// TwinCAT 3 PLC project TwinCAT_OpenFramework_Loggers
// Title: TwinCAT Open Framework Loggers
// Company: Oleksandr Tiutyk FOP
// Author: Oleksandr Tiutyk
// ProjectVersion: 1.0.13.0
// Description: Various loggers implementation for TwinCAT.OpenFramework
// ProgramVersion: 3.1.4026.28
// libraries:
//   Tc2_Standard, * (Beckhoff Automation GmbH)
//   Tc2_System, * (Beckhoff Automation GmbH)
//   Tc2_Utilities, * (Beckhoff Automation GmbH)
//   Tc3_EventLogger, * (Beckhoff Automation GmbH)
//   Tc3_Module, * (Beckhoff Automation GmbH)
//   [TwinCAT Open Framework Collections], * (Oleksandr Tiutyk FOP)
//   [TwinCAT Open Framework Core], * (Oleksandr Tiutyk FOP)
//   [TwinCAT Open Framework File System], * (Oleksandr Tiutyk FOP)
// project tree:
//   QueuedLogger/ QueuedLogger.TcPOU, QUEUED_LOG_MESSAGE.TcDUT
//   / Parameters.TcGVL
//   EventLogger/ EventLogger.TcPOU
//   FileLogger/ SimpleTextFileLogger.TcPOU, SIMPLE_TEXT_FILE_LOGGER_STATE.TcDUT
//   Internal/ CurrentNamespace.TcPOU, NamespaceExtractor.TcPOU
//   Version/ Global_Version.TcGVL
// (motion and I/O tree: see PLC project twincat_openframework_core)
// real-time tasks:
//   TASK PlcTask: cycle T#10ms, priority 20, ADS port 350
//   TASK TestTask: cycle T#10ms, priority 1, ADS port 351
//   TASK RunnerTestTask: cycle T#10ms, priority 2, ADS port 354
//   TASK HowToTask: cycle T#10ms, priority 22, ADS port 353
// variable links:

// ---- QueuedLogger/QUEUED_LOG_MESSAGE.TcDUT
(*
SPDX-FileCopyrightText: © 2026 Oleksandr Tiutyk <trofimich@gmail.com>
SPDX-License-Identifier: MIT
License: https://opensource.org/license/mit
*)

(*!
<summary>Stores an owned text snapshot waiting for a logging backend.</summary>
<description>
Internal QueuedLogger storage. Text, category and optional number are copied by value. Contains no borrowed
references to caller data or exceptions.
</description>
*)
TYPE QUEUED_LOG_MESSAGE :
STRUCT
	Message : TOF_Core.ERROR_MESSAGE;
	Category : TOF_Core.LOG_CATEGORY;
	HasMessageNumber : BOOL;
	MessageNumber : ULINT;
END_STRUCT
END_TYPE

// ---- FileLogger/SIMPLE_TEXT_FILE_LOGGER_STATE.TcDUT
(*!
<summary>Identifies the current phase of a text-file logger.</summary>
<description>
Stop first drains accepted messages in the current initialization/logging phase. STOPPING then advances final
file release; STOPPED permits explicit Start. FAILED remains terminal and may still require cyclic cleanup.
New states follow FAILED so the existing state ordinals remain unchanged.
</description>
*)
{attribute 'qualified_only'}
{attribute 'strict'}
{attribute 'to_string'}
TYPE SIMPLE_TEXT_FILE_LOGGER_STATE :
(
	INITIAL,
	CREATING_DIRECTORY, 
	LOGGING, 
	FAILED,
	STOPPING,
	STOPPED
);
END_TYPE

// ---- Parameters.TcGVL
(*
SPDX-FileCopyrightText: © 2026 Oleksandr Tiutyk <trofimich@gmail.com>
SPDX-License-Identifier: MIT
License: https://opensource.org/license/mit
*)

(*!
<summary>Provides configurable library limits for logging.</summary>
<description>Limits apply independently to each logger instance, not to a shared memory budget.</description>
*)
{attribute 'qualified_only'}
VAR_GLOBAL CONSTANT
	(*!
	<summary>Maximum number of messages waiting in each SimpleTextFileLogger message queue.</summary>
	<description>
	When the queue reaches this limit, TryLog methods return FALSE before formatting or allocating queued text.
	Already accepted messages are retained. The current send batch is excluded and is limited separately by
	maxRecordsPerFile. Zero prevents acceptance of new messages.
	</description>
	*)
	MAX_PENDING_LOG_MESSAGES : UINT := 50;

	(*!
	<summary>Maximum number of text records waiting in each QueuedLogger.</summary>
	<description>
	Fixed per-instance storage; each record includes an ERROR_MESSAGE and number metadata. The array reserves one
	extra slot so zero capacity is representable; zero rejects all records. One additional record is reserved for
	the active backend call. Capacity also bounds records forwarded by one Execute. Full queues reject new
	records without waiting for free space; acquiring the queue lock may still block.
	</description>
	*)
	QUEUED_LOGGER_CAPACITY : UINT := 100;
END_VAR

// ---- Version/Global_Version.TcGVL
{attribute 'TcGenerated'}
{attribute 'no-analysis'}
{attribute 'linkalways'}
// This function has been automatically generated from the project information.
VAR_GLOBAL CONSTANT
	{attribute 'const_non_replaced'}
	stLibVersion_TwinCAT_Open_Framework_Loggers : ST_LibVersion := (iMajor := 1, iMinor := 0, iBuild := 13, iRevision := 0, nFlags := 0, sVersion := '1.0.13.0');
END_VAR

// ---- FileLogger/SimpleTextFileLogger.TcPOU
(*
SPDX-FileCopyrightText: © 2026 Oleksandr Tiutyk <trofimich@gmail.com>
SPDX-License-Identifier: MIT
License: https://opensource.org/license/mit
*)

(*!
<summary>Formats diagnostics for text-file logging and advances file operations through cyclic execution.</summary>
<description>
Use this backend for buffered text-file output. Direct TryLog and Execute calls on one instance must belong to
one task: its message queue, buffers and file-operation state are not synchronized for concurrent access. For
callers in multiple tasks, use QueuedLogger and let its owner task service this backend; do not bypass the
wrapper with concurrent direct calls. Separate instances writing independently must use separate output files.
Cyclic Execute is required to advance writing and cleanup. Exception logging accepts IReadOnlyException and
reads borrowed diagnostics without transferring ownership. Implementations must not retain exception
references beyond their task cleanup. FAILED is terminal for this instance: no automatic retry or recovery is
provided. Continue calling Execute after failure to discard queued messages, cancel active tasks and release
the send buffer once file operations have finished. Pending messages are not retried. The instance must remain
alive during cleanup. Busy reports pending initialization, messages, file operations or failure cleanup; an
idle open file alone does not make it TRUE. Busy = FALSE does not mean the file handle is closed. After Stop
or in FAILED state, or when the per-instance message queue reaches Parameters.MAX_PENDING_LOG_MESSAGES, all
TryLog methods return FALSE before formatting or queuing new diagnostics. Full-queue rejection preserves
already accepted messages; the current send batch is separate from this limit. Buffered text preserves the
optional message number and category prefix; oversized text is truncated to ERROR_MESSAGE capacity with a
final ellipsis. TryLog methods and Execute do not propagate exceptions. Failed admission returns FALSE;
Execute failures enter FAILED and require further cleanup calls. The terminal allocation latch is preserved
for the task boundary. The initial instance starts automatically through Execute. Stop requests draining of
accepted messages and best-effort file release; continue Execute until STOPPED or until FAILED cleanup
finishes. Start resumes only STOPPED, retaining the file counter and opening the next generated file when a
message arrives. New messages are rejected from Stop until Start. Lifecycle calls belong to the same owner
task as Execute. STOPPED means the close attempt and buffer cleanup finished, not certified physical closure
after a native close error; the underlying resource manager retains its best-effort policy. Embedded task
and resource diagnostics use an owned AdsLogger directly, bypassing LogManager filters/counters and avoiding
feedback into this logger or its QueuedLogger wrapper. maxRecordsPerFile must be positive; zero rejects
admission and the first Execute enters FAILED before any filesystem operation. The configured timeout
applies to directory, open, write and close requests, not to the whole logger lifecycle.
</description>
*)

{attribute 'no_explicit_call' := 'do not call this function block directly'}
FUNCTION_BLOCK SimpleTextFileLogger EXTENDS TOF_Core.Object IMPLEMENTS TOF_Core.ILogger
VAR_STAT
	//! <summary>Static type metadata shared by instances without reading mutable instance state.</summary>
	_ClassName : STRING := __POUNAME();
END_VAR
VAR
	
	{attribute 'hide'} 
	_State : SIMPLE_TEXT_FILE_LOGGER_STATE;
	{attribute 'hide'} 
	_ErrorMessage : TOF_Core.ERROR_MESSAGE;
	{attribute 'hide'}
	_CleanupPending : BOOL;

	//!<summary>
	//! Blocks new messages while accepted work drains and remains set until Start resumes a stopped logger.
	//! </summary>
	_StopRequested : BOOL;
	
	_LogFilePrefix : STRING(32);

	//! <summary>Independent owner-task channel for embedded task and file-resource diagnostics.</summary>
	_InternalDiagnosticLogger : TOF_Core.AdsLogger;

	_CreateDirectoryIfNotExists : TOF_FileSystem.CreateDirectoryIfNotExists(name := "CreateDirectoryIfNotExists");	
	
	_FileContentManager : TOF_FileSystem.FileContentManager(name := "FileContentManager");
	_RecordsPerFile : UINT;
	_WriteBytesTask : TOF_FileSystem.WriteBytesToFile(name := "WriteBytesTask");
	
	_MaxRecordsPerFile : UINT := 100;
	
	_Queue : ARRAY [0..Parameters.MAX_PENDING_LOG_MESSAGES - 1] OF TOF_Core.ERROR_MESSAGE;
	_ReadIndex : UDINT;
	_WriteIndex : UDINT;
	_QueueCount : UDINT;

	_SendBuffer : TOF_Collections.ByteList<0>;
	
	_LogFileCounter : UDINT;
END_VAR

(*!
<summary>Reports the ADS target copied at construction.</summary>
<description>
Directory and file operations use this target; an empty value selects the local system. No I/O is performed.
</description>
*)
{attribute 'monitoring' := 'call'}
PROPERTY AmsNetId : Tc2_System.T_AmsNetID
GET
AmsNetId := _CreateDirectoryIfNotExists.AmsNetId;
END_GET
END_PROPERTY

(*!
<summary>Reports unfinished initialization, message processing, file operations or failure cleanup.</summary>
<description>
TRUE before initialization finishes, while messages or file tasks remain pending, during file acquisition or
release, while a requested normal stop is unfinished, and until failure cleanup completes. An open file
waiting for new messages does not make the logger busy. FALSE does not certify successful writes or a closed
file handle. Continue Execute while cleanup is pending after FAILED.
</description>
*)
{attribute 'monitoring' := 'call'}
PROPERTY Busy : BOOL
GET
Busy := _State = SIMPLE_TEXT_FILE_LOGGER_STATE.INITIAL
	OR_ELSE _State = SIMPLE_TEXT_FILE_LOGGER_STATE.CREATING_DIRECTORY
	OR_ELSE (_StopRequested
		AND_THEN _State <> SIMPLE_TEXT_FILE_LOGGER_STATE.STOPPED
		AND_THEN _State <> SIMPLE_TEXT_FILE_LOGGER_STATE.FAILED)
	OR_ELSE _CleanupPending
	OR_ELSE _QueueCount > TOF_Core.UnsignedInt32.ZERO
	OR_ELSE _FileContentManager.PendingTaskCount > 0
	OR_ELSE _WriteBytesTask.State.Running
	OR_ELSE _WriteBytesTask.FileOperationInProgress
	OR_ELSE (_FileContentManager.State.Running AND_THEN NOT _FileContentManager.RunningSubstate.Processing);
END_GET
END_PROPERTY

(*!
<summary>Provides the concrete logger type name.</summary>
<description>
Returns borrowed read-only initialized static storage. Reading has no side effects or exceptions.
Do not modify the referenced metadata; initialized storage is available before base initialization.
</description>
*)
{attribute 'monitoring' := 'call'}
PROPERTY ClassName : REFERENCE TO STRING
GET
ClassName REF= _ClassName;
END_GET
END_PROPERTY

(*!
<summary>Builds the current log path from the configured directory, prefix, local timestamp and file counter.</summary>
<description>
Uses the existing naming policy without checking for an existing file. A path that exceeds the return capacity
raises StringOverflowException for Execute to report as FAILED. Computes the path on the stack without dynamic
string-builder allocations; no truncated path is used.
</description>
*)
METHOD PRIVATE createCurrentFilePath : Tc2_System.T_MaxString
VAR
	directoryPathText : Tc2_System.T_MaxString;
	timestampText : STRING(32);
	counterText : STRING(16);
	filePathLength : UDINT;
END_VAR
directoryPathText := DirectoryPath;
timestampText := TOF_Core.DateAndTimes.ToString(value := LDT_TO_DT(TOF_Core.System.SystemLocalDateTime));
counterText := TO_STRING(_LogFileCounter);

// Fixed separators and extension '\' + '_' + '_' + '.log' add 7 characters.
filePathLength := TO_UDINT(Tc2_Standard.LEN(STR := directoryPathText))
	+ TO_UDINT(Tc2_Standard.LEN(STR := _LogFilePrefix))
	+ TO_UDINT(Tc2_Standard.LEN(STR := timestampText))
	+ TO_UDINT(Tc2_Standard.LEN(STR := counterText))
	+ 7;

IF filePathLength > 255 THEN
	TOF_Core.Exceptions.ThrowStringOverflow(
		sourceNamespaceName := NamespaceName,
		sourceClassName := ClassName,
		sourcePOUName := __POUNAME(),
		sourcePosition := __POSITION(),
		stringName := 'CurrentFilePath',
		actualLength := filePathLength,
		maxLength := 255
	);  
END_IF

createCurrentFilePath := TOF_Core.Strings.Concat255(
	directoryPathText,
	'\',
	_LogFilePrefix,
	'_',
	timestampText,
	'_',
	counterText,
	'.log');
END_METHOD

(*!
<summary>Reports the copied output directory.</summary>
<description>
The native target resolves this path with DirectoryPathType. Filename generation retains the configured
directory and rejects overflow rather than silently truncating the generated path.
</description>
*)
{attribute 'monitoring' := 'call'}
PROPERTY DirectoryPath : Tc2_System.T_MaxString
GET
DirectoryPath := _CreateDirectoryIfNotExists.DirectoryPath;
END_GET
END_PROPERTY

(*!
<summary>Reports the native path context copied at construction.</summary>
<description>
Used by both directory creation and file opening; this observation does not validate or open a path.
</description>
*)
{attribute 'monitoring' := 'call'}
PROPERTY DirectoryPathType : Tc2_System.E_OpenPath
GET
DirectoryPathType := _CreateDirectoryIfNotExists.PathType;
END_GET
END_PROPERTY

(*!
<summary>Borrows the retained terminal failure diagnostic.</summary>
<description>
Meaningful after State becomes FAILED; cleanup preserves the original diagnostic. The reference remains
valid while this instance lives. Treat it as read-only: ST reference assignment can otherwise mutate it.
Read only from the logger owner task or with external synchronization; no cross-task snapshot is provided.
</description>
*)
{attribute 'monitoring' := 'call'}
PROPERTY ErrorMessage : REFERENCE TO TOF_Core.ERROR_MESSAGE
GET
ErrorMessage REF= _ErrorMessage;
END_GET
END_PROPERTY

(*!
<summary>Advances initialization, writing, requested normal stopping or cleanup after terminal failure.</summary>
<description>
Does not propagate exceptions. On the first failure, enters FAILED and attempts to store the diagnostic. If
diagnostic extraction fails, stores a fixed fallback message without allocating an exception. Subsequent calls
discard queued messages and advance cancellation without starting new writes. The send buffer is released only
after its task and file operation have finished and the manager is no longer running. Cleanup exceptions are
caught; cleanup remains pending for a later call without replacing the original ErrorMessage or recovering the
logger. Fatal allocation state remains latched for the task boundary. After Stop, initialization and already
accepted messages finish normally, including file rotation. Once all writes complete, STOPPING advances
resource release without scheduling further messages. Only then are the manager and write task reset and the
send buffer released before entering STOPPED. A failure during draining uses the existing FAILED path and may
discard unwritten messages. Execute does nothing in STOPPED; Start is required to resume.
</description>
*)
METHOD Execute
VAR	
	exceptionCode : __SYSTEM.ExceptionCode;
	exception : TOF_Core.IException;
END_VAR
VAR
	formattedExceptionMessage : TOF_Core.ERROR_MESSAGE;
END_VAR
__TRY
	stopAfterAllocationFailure();

	IF _State = SIMPLE_TEXT_FILE_LOGGER_STATE.INITIAL
		AND_THEN _MaxRecordsPerFile = TOF_Core.UnsignedInt16.MIN_VALUE
	THEN
		_ErrorMessage := "MaxRecordsPerFile must be greater than zero.";
		_State := SIMPLE_TEXT_FILE_LOGGER_STATE.FAILED;
		_CleanupPending := TRUE;
	END_IF

	IF _State = SIMPLE_TEXT_FILE_LOGGER_STATE.FAILED THEN

		IF NOT _CleanupPending THEN
			RETURN;
		END_IF

		_QueueCount := 0;
		_ReadIndex := 0;
		_WriteIndex := 0;

		IF _CreateDirectoryIfNotExists.State.Running THEN
			_CreateDirectoryIfNotExists.Cancel();
			_CreateDirectoryIfNotExists.Execute();
		END_IF

		IF _FileContentManager.State.Running THEN
			_FileContentManager.Cancel();
			_FileContentManager.Execute();
		END_IF

		IF NOT _CreateDirectoryIfNotExists.State.Running
			AND_THEN NOT _FileContentManager.State.Running
			AND_THEN NOT _WriteBytesTask.State.Running
			AND_THEN NOT _WriteBytesTask.FileOperationInProgress
		THEN
			_FileContentManager.ClearWaitingTasks();

			_WriteBytesTask.SourceBuffer := 0;
			_WriteBytesTask.BytesCountToWrite := 0;
			_SendBuffer.Clear(releaseDynamicMemory := TRUE);
			_CleanupPending := FALSE;
		END_IF

		RETURN;
	END_IF

	CASE _State OF
		SIMPLE_TEXT_FILE_LOGGER_STATE.INITIAL:

			IF _StopRequested AND_THEN _QueueCount = TOF_Core.UnsignedInt32.ZERO THEN
				_State := SIMPLE_TEXT_FILE_LOGGER_STATE.STOPPED;
				RETURN;
			END_IF

			_CreateDirectoryIfNotExists.Reset();

			IF stopAfterAllocationFailure() THEN
				RETURN;
			END_IF

			_CreateDirectoryIfNotExists.Start();

			IF stopAfterAllocationFailure() THEN
				RETURN;
			END_IF

			_State := SIMPLE_TEXT_FILE_LOGGER_STATE.CREATING_DIRECTORY;

		SIMPLE_TEXT_FILE_LOGGER_STATE.CREATING_DIRECTORY:
			_CreateDirectoryIfNotExists.Execute();

			IF stopAfterAllocationFailure() THEN
				RETURN;
			END_IF

			IF _CreateDirectoryIfNotExists.State.Stopped THEN

				IF _CreateDirectoryIfNotExists.FinalStopReason.WorkDone THEN
					_State := SIMPLE_TEXT_FILE_LOGGER_STATE.LOGGING;
				ELSE
					TOF_Core.Exceptions.ThrowStandard(
						sourceNamespaceName := NamespaceName,
						sourceClassName := ClassName,
						sourcePOUName := __POUNAME(),
						sourcePosition := __POSITION(),
						message := "Log directory not created"
					);
				END_IF

			END_IF

		SIMPLE_TEXT_FILE_LOGGER_STATE.LOGGING:
			_FileContentManager.Execute();

			IF stopAfterAllocationFailure() THEN
				RETURN;
			END_IF

			IF _FileContentManager.State.Stopped AND_THEN _FileContentManager.FinalStopReason.Failure THEN
				formattedExceptionMessage := _FileContentManager.FinalStopReason.Message;

				TOF_Core.Exceptions.ThrowStandard(
					sourceNamespaceName := NamespaceName,
					sourceClassName := ClassName,
					sourcePOUName := __POUNAME(),
					sourcePosition := __POSITION(),
					message := formattedExceptionMessage
				);
			END_IF

			processPendingMessages();

			IF stopAfterAllocationFailure() THEN
				RETURN;
			END_IF

			IF _StopRequested
				AND_THEN _QueueCount = TOF_Core.UnsignedInt32.ZERO
				AND_THEN _FileContentManager.PendingTaskCount = TOF_Core.SignedInt32.ZERO
			THEN
				_FileContentManager.StopWhenNoPendingTasks := TRUE;
				_State := SIMPLE_TEXT_FILE_LOGGER_STATE.STOPPING;
			END_IF

		SIMPLE_TEXT_FILE_LOGGER_STATE.STOPPING:
			_FileContentManager.Execute();

			IF stopAfterAllocationFailure() THEN
				RETURN;
			END_IF

			IF _FileContentManager.State.Stopped AND_THEN _FileContentManager.FinalStopReason.Failure THEN
				_ErrorMessage := _FileContentManager.FinalStopReason.Message;
				_State := SIMPLE_TEXT_FILE_LOGGER_STATE.FAILED;
				_CleanupPending := TRUE;
				RETURN;
			END_IF

			IF NOT _FileContentManager.State.Running THEN
				(* No queued write or native I/O remains; borrowed buffer storage may now be released. *)
				_FileContentManager.Reset();

				IF stopAfterAllocationFailure() THEN
					RETURN;
				END_IF

				_FileContentManager.StopWhenNoPendingTasks := FALSE;
				_WriteBytesTask.Reset();

				IF stopAfterAllocationFailure() THEN
					RETURN;
				END_IF

				_WriteBytesTask.SourceBuffer := TOF_Core.Memory.NULL_ADDRESS;
				_WriteBytesTask.BytesCountToWrite := TOF_Core.UnsignedInt32.ZERO;
				_SendBuffer.Clear(releaseDynamicMemory := TRUE);
				_RecordsPerFile := 0;

				_State := SIMPLE_TEXT_FILE_LOGGER_STATE.STOPPED;
			END_IF

	END_CASE

__CATCH(exceptionCode)
	IF _State <> SIMPLE_TEXT_FILE_LOGGER_STATE.FAILED THEN
		_State := SIMPLE_TEXT_FILE_LOGGER_STATE.FAILED;
		_CleanupPending := TRUE;

		__TRY
			exception := TOF_Core.ExceptionManager.GetLastException(
				exceptionCode := exceptionCode,
				catchPointNamespaceName := NamespaceName,
				catchPointPOUName := __POUNAME(),
				catchPointPosition := __POSITION()
			);
			_ErrorMessage := exception.GetMessage();
		__CATCH
			_ErrorMessage := "File logger failed; diagnostic information is unavailable.";
		__ENDTRY

	END_IF

__ENDTRY
END_METHOD

(*!
<summary>Copies logger configuration and binds an independent diagnostic route without performing I/O.</summary>
<description>
All additional constructor arguments must be supplied explicitly. directoryPath and logFilePrefix determine
the existing timestamp/counter filename policy; instances must use separate output files. maxRecordsPerFile
must be positive. Zero is retained without throwing here; TryLog rejects it and Execute reports FAILED before
filesystem I/O. timeout applies to directory, open, write and close requests. Lifecycle initialization only
copies configuration and borrowed routes; it does not create exceptions or invoke diagnostic callbacks.
</description>
<param name="directoryPath">Output directory resolved on the configured ADS target.</param>
<param name="logFilePrefix">Filename prefix copied for this instance.</param>
<param name="maxRecordsPerFile">Positive record count; zero is reported by Execute before I/O.</param>
<param name="directoryPathType">Native path context for directory and file operations.</param>
<param name="timeout">Per-request native timeout for directory, open, write and close.</param>
<param name="amsNetId">ADS target; empty selects the local system.</param>
*)
METHOD FB_init : BOOL
VAR_INPUT
	bInitRetains : BOOL; // TRUE: the retain variables are initialized (reset warm / reset cold)
	bInCopyCode : BOOL;  // TRUE: the instance will be copied to the copy code afterward (online change)
	directoryPath : Tc2_System.T_MaxString;
	logFilePrefix : STRING(32);
	maxRecordsPerFile : UINT;
	directoryPathType : Tc2_System.E_OpenPath; 
	timeout : TIME; 
	amsNetId : Tc2_System.T_AmsNetID; 
END_VAR
_CreateDirectoryIfNotExists.DiagnosticLogger := _InternalDiagnosticLogger;
_FileContentManager.DiagnosticLogger := _InternalDiagnosticLogger;
_WriteBytesTask.DiagnosticLogger := _InternalDiagnosticLogger;
_WriteBytesTask.Timeout := timeout;

_CreateDirectoryIfNotExists.DirectoryPath := directoryPath;
_CreateDirectoryIfNotExists.PathType := directoryPathType;
_CreateDirectoryIfNotExists.Timeout := timeout;
_CreateDirectoryIfNotExists.AmsNetId := amsNetId;

_FileContentManager.PathType := directoryPathType;
_FileContentManager.ModeFlags := Tc2_System.Global_Variables.FOPEN_MODEWRITE
	OR Tc2_System.Global_Variables.FOPEN_MODEPLUS
	OR Tc2_System.Global_Variables.FOPEN_MODETEXT;
_FileContentManager.Timeout := timeout;
_FileContentManager.AmsNetId := amsNetId;

_LogFilePrefix := logFilePrefix;

_MaxRecordsPerFile := maxRecordsPerFile;
END_METHOD

(*!
<summary>Reports the filename prefix copied at construction.</summary>
<description>
Combined with local timestamp and the retained counter; it does not establish exclusive creation or
global uniqueness. Use separate output files for independent logger instances.
</description>
*)
{attribute 'monitoring' := 'call'}
PROPERTY LogFilePrefix : STRING(32)
GET
LogFilePrefix := _LogFilePrefix;
END_GET
END_PROPERTY

(*!
<summary>Reports the positive number of diagnostic records permitted in one generated file.</summary>
<description>
Zero is a configuration error: TryLog rejects admission and Execute records FAILED before filesystem I/O.
The limit counts diagnostic records, not physical lines inside a message; rotation advances on Execute.
</description>
*)
{attribute 'monitoring' := 'call'}
PROPERTY MaxRecordsPerFile : UINT
GET
MaxRecordsPerFile := _MaxRecordsPerFile;
END_GET
END_PROPERTY

(*!
<summary>Borrows the library namespace.</summary>
<description>
Read-only compiler-initialized namespace storage; do not modify the referenced text.
</description>
*)
{attribute 'monitoring' := 'call'}
PROPERTY NamespaceName : REFERENCE TO STRING
GET
NamespaceName REF= CurrentNamespace.Name;
END_GET
END_PROPERTY

(*!
<summary>Transfers queued messages into a batch and schedules its asynchronous file write.</summary>
<description>
Called by Execute. Leaves messages queued while a previous file task or file rotation is pending. Removes
messages from the queue as they are copied into the send buffer, up to the per-file record limit. The send
buffer must remain alive until the write operation finishes. Invalid write-task state and failures from nested
operations propagate to Execute for its failure handling and cleanup. Returning does not mean that the
messages have been written to the file.
</description>
*)
METHOD PRIVATE processPendingMessages
VAR
	formattedExceptionMessage : TOF_Core.ERROR_MESSAGE;
END_VAR
IF _QueueCount = 0 OR_ELSE _FileContentManager.PendingTaskCount > 0 THEN
	RETURN;
END_IF

IF NOT _WriteBytesTask.State.Ready AND_THEN NOT _WriteBytesTask.State.Stopped THEN
	formattedExceptionMessage := TOF_Core.WideStrings.Concat255(
		"WriteBytesTask has invalid state '",
		TO_WSTRING(_WriteBytesTask.State.Value),
		"'"
	);

	TOF_Core.Exceptions.ThrowStandard(
		sourceNamespaceName := NamespaceName,
		sourceClassName := ClassName,
		sourcePOUName := __POUNAME(),
		sourcePosition := __POSITION(),
		message := formattedExceptionMessage
	);
END_IF

IF _WriteBytesTask.State.Stopped AND_THEN NOT _WriteBytesTask.FinalStopReason.WorkDone THEN
	formattedExceptionMessage := TOF_Core.WideStrings.Concat255(
		"WriteBytesTask has invalid stop reason '",
		TO_WSTRING(_WriteBytesTask.FinalStopReason.Value),
		"'"
	);

	TOF_Core.Exceptions.ThrowStandard(
		sourceNamespaceName := NamespaceName,
		sourceClassName := ClassName,
		sourcePOUName := __POUNAME(),
		sourcePosition := __POSITION(),
		message := formattedExceptionMessage
	);
END_IF

IF _RecordsPerFile >= _MaxRecordsPerFile AND_THEN _FileContentManager.State.Running THEN

	IF NOT _FileContentManager.RunningSubstate.ResourceReleasing THEN
		_FileContentManager.Cancel();
	END_IF

	IF _FileContentManager.State.Running THEN
		RETURN;
	END_IF

END_IF

_SendBuffer.Clear();

IF _FileContentManager.FilePath = '' OR_ELSE _RecordsPerFile >= _MaxRecordsPerFile THEN
	_RecordsPerFile := 0;
	_LogFileCounter := _LogFileCounter + 1;

	_FileContentManager.Reset();

	IF stopAfterAllocationFailure() THEN
		RETURN;
	END_IF

	_FileContentManager.FilePath := createCurrentFilePath();

	_FileContentManager.Start();

	IF stopAfterAllocationFailure() THEN
		RETURN;
	END_IF

	_SendBuffer.AppendData(
		data := ADR(TOF_Core.WideStrings.ByteOrderMark),
		dataSize := SIZEOF(TOF_Core.WideStrings.ByteOrderMark)
	);
END_IF

WHILE _QueueCount > 0 DO
	_SendBuffer.AppendData(
		data := ADR(_Queue[_ReadIndex]),
		dataSize := TO_DINT(Tc2_Utilities.WLEN2(pWSTRING := ADR(_Queue[_ReadIndex])) * TOF_Core.WideStrings.CharSize)
	);
	_SendBuffer.AppendData(
		data := ADR(TOF_Core.WideStrings.NewLine),
		dataSize := TO_DINT(SIZEOF(TOF_Core.WideStrings.NewLine) - TOF_Core.WideStrings.CharSize)
	);

	_ReadIndex := _ReadIndex + 1;

	IF _ReadIndex >= Parameters.MAX_PENDING_LOG_MESSAGES THEN
		_ReadIndex := 0;
	END_IF

	_QueueCount := _QueueCount - 1;

	_RecordsPerFile := _RecordsPerFile + 1;

	IF _RecordsPerFile >= _MaxRecordsPerFile THEN
		EXIT;
	END_IF

END_WHILE

_WriteBytesTask.Reset();

IF stopAfterAllocationFailure() THEN
	RETURN;
END_IF

_WriteBytesTask.SourceBuffer := _SendBuffer.DataAddress;
_WriteBytesTask.BytesCountToWrite := TO_UDINT(_SendBuffer.Length);

_FileContentManager.Enqueue(fileHandleTask := _WriteBytesTask);
END_METHOD

(*!
<summary>Reports the size of the concrete logger instance in bytes.</summary>
<description>
Includes the fixed queue and embedded instances; separately allocated dynamic buffers are excluded.
</description>
*)
{attribute 'monitoring' := 'call'}
PROPERTY SelfSize : ULINT
GET
SelfSize := XSIZEOF(THIS^);
END_GET
END_PROPERTY

(*!
<summary>Resumes a normally stopped logger and permits new messages.</summary>
<description>
Call from the owner task. Returns TRUE only from STOPPED; INITIAL already starts automatically, and
initializing, logging, stopping or FAILED instances return FALSE without changing state. Does not perform I/O
or propagate exceptions. Subsequent Execute calls check the directory again. The next accepted message opens
the next generated file using the retained counter, rather than reopening the previous file. This uses the
existing naming policy, not exclusive creation or global name uniqueness. Does not recover a FAILED instance
or certify that an earlier best-effort close succeeded.
</description>
*)
METHOD Start : BOOL
IF _State <> SIMPLE_TEXT_FILE_LOGGER_STATE.STOPPED THEN
	RETURN;
END_IF

_StopRequested := FALSE;
_State := SIMPLE_TEXT_FILE_LOGGER_STATE.INITIAL;
Start := TRUE;
END_METHOD

(*!
<summary>Reports initialization, logging, normal stopping, stopped or terminal failure state.</summary>
<description>
After Stop, the current initialization/logging state persists while accepted messages drain; STOPPING then
denotes final file release. STOPPED permits Start and has no pending writes or buffer cleanup, but does not
certify physical closure after a native close error. FAILED does not recover automatically and rejects new
diagnostics. It does not by itself certify that pending file operations have finished or buffered memory has
been released.
</description>
*)
{attribute 'monitoring' := 'call'}
PROPERTY State : SIMPLE_TEXT_FILE_LOGGER_STATE
GET
State := _State;
END_GET
END_PROPERTY

(*!
<summary>Requests completion of accepted messages followed by normal file release.</summary>
<description>
Call from the owner task. Returns TRUE for an accepted or repeated request, including STOPPED. Returns FALSE
in FAILED, where Execute must instead finish the existing failure cleanup. Immediately rejects new TryLog
calls without discarding accepted messages. Does not perform I/O or propagate exceptions. Continue cyclic
Execute until STOPPED; failures may enter FAILED and discard unwritten messages under its existing cleanup
policy. Start cannot cancel an unfinished stop. Best-effort close completion is not a guarantee of physical
release after a native close error.
</description>
*)
METHOD Stop : BOOL
IF _State = SIMPLE_TEXT_FILE_LOGGER_STATE.FAILED THEN
	RETURN;
END_IF

_StopRequested := TRUE;
Stop := TRUE;
END_METHOD

(*!
<summary>Reports the per-request native timeout copied at construction.</summary>
<description>
Applies to directory enumeration/creation and file open, write and close requests. It is not a deadline
for the whole logger lifecycle or a guarantee of physical release after native failure.
</description>
*)
{attribute 'monitoring' := 'call'}
PROPERTY Timeout : TIME
GET
Timeout := _CreateDirectoryIfNotExists.Timeout;
END_GET
END_PROPERTY

(*!
<summary>Formats an error and queues its text for later file writing.</summary>
<description>
Returns FALSE after Stop or in FAILED state, or when the message queue is full before reading or formatting
the error. An invalid reference is ignored. Otherwise delegates to TryLogMessage; TRUE confirms buffering, not
completion of the file write. Exceptions are caught and reported as FALSE without further logging. The
terminal allocation latch is preserved.
Returns FALSE when fatal allocation state is observed before work or after nested calls. The latch remains
set for the caller's task boundary; already accepted or emitted records are not rolled back.
</description>
<param name="error">Borrowed error to format.</param>
<param name="messageNumber">Optional borrowed number to include in the buffered text.</param>
*)
METHOD TryLogError : BOOL
VAR_INPUT
	error : REFERENCE TO TOF_Core.ERROR;
	messageNumber : REFERENCE TO ULINT := 0;
END_VAR
VAR
	message : TOF_Core.ERROR_MESSAGE;
END_VAR
__TRY

	IF TOF_Core.DynamicMemoryManager.HasAllocationFailed THEN
		RETURN;
	END_IF

	IF _MaxRecordsPerFile = TOF_Core.UnsignedInt16.MIN_VALUE
		OR_ELSE _StopRequested
		OR_ELSE _State = SIMPLE_TEXT_FILE_LOGGER_STATE.FAILED
		OR_ELSE _QueueCount >= Parameters.MAX_PENDING_LOG_MESSAGES
	THEN
		TryLogError := FALSE;
		RETURN;
	END_IF

	IF NOT __ISVALIDREF(error) THEN
		RETURN;
	END_IF

	message := error.ToString(
		sourceDisplayMode := TOF_Core.ERROR_SOURCE_DISPLAY_MODE.HIDDEN,
		timestampDisplayMode := TOF_Core.TIMESTAMP_DISPLAY_MODE.LOCAL
	);

	TryLogError := TryLogMessage(
		category := SEL(
			error.Severity = TOF_Core.ERROR_SEVERITY.CRITICAL,
			TOF_Core.LOG_CATEGORY.ERROR,
			TOF_Core.LOG_CATEGORY.CRITICAL_ERROR
		),
		message := message,
		messageNumber := messageNumber
	);

	IF TOF_Core.DynamicMemoryManager.HasAllocationFailed THEN
		TryLogError := FALSE;
	END_IF

__CATCH
	TryLogError := FALSE;
__ENDTRY
END_METHOD

(*!
<summary>Attempts to log diagnostic information from a read-only exception view.</summary>
<description>
Borrows the exception for the call without clearing it or taking ownership. The exception and its inner causes
must remain live while their diagnostics are read. Logging does not extend their lifetime. Returns FALSE after
Stop or in FAILED state, or when the message queue is full before reading or formatting the exception.
Otherwise TRUE confirms buffering, not completion of the file write. Exceptions are caught and reported as
FALSE without further logging. The terminal allocation latch is preserved.
Returns FALSE when fatal allocation state is observed before work or after nested calls. The latch remains
set for the caller's task boundary; already accepted or emitted records are not rolled back.
</description>
<param name="exception">Exception view to read; null is ignored.</param>
<param name="severity">Severity used to select the log category.</param>
*)
METHOD TryLogException : BOOL
VAR_INPUT
	exception : TOF_Core.IReadOnlyException;
	severity : TOF_Core.ERROR_SEVERITY;
	messageNumber : REFERENCE TO ULINT := 0;
END_VAR
VAR
	message : TOF_Core.ERROR_MESSAGE;
END_VAR
__TRY

	IF TOF_Core.DynamicMemoryManager.HasAllocationFailed THEN
		RETURN;
	END_IF

	IF _MaxRecordsPerFile = TOF_Core.UnsignedInt16.MIN_VALUE
		OR_ELSE _StopRequested
		OR_ELSE _State = SIMPLE_TEXT_FILE_LOGGER_STATE.FAILED
		OR_ELSE _QueueCount >= Parameters.MAX_PENDING_LOG_MESSAGES
	THEN
		TryLogException := FALSE;
		RETURN;
	END_IF

	IF exception = 0 THEN
		RETURN;
	END_IF

	message := exception.GetMessage(showSource := TRUE, timestampDisplayMode := TOF_Core.TIMESTAMP_DISPLAY_MODE.LOCAL);

	TryLogException := TryLogMessage(
		category := SEL(severity = TOF_Core.ERROR_SEVERITY.CRITICAL, TOF_Core.LOG_CATEGORY.ERROR, TOF_Core.LOG_CATEGORY.CRITICAL_ERROR),
		message := message,
		messageNumber := messageNumber
	);

	IF TOF_Core.DynamicMemoryManager.HasAllocationFailed THEN
		TryLogException := FALSE;
	END_IF

__CATCH
	TryLogException := FALSE;
__ENDTRY
END_METHOD

(*!
<summary>Formats a diagnostic and queues its text for later file writing.</summary>
<description>
Returns FALSE after Stop or in FAILED state, or when the queue reaches Parameters.MAX_PENDING_LOG_MESSAGES,
before formatting or allocating buffered text. Queue rejection does not discard previously accepted messages.
Otherwise formats an optional message number followed by the category and message. Preserves the prefixes and
marks truncated text with an ellipsis. Formatting uses local storage without raising a size-overflow
exception. Text admission copies into fixed instance-owned queue storage without heap allocation. Returns TRUE after successful insertion
into the message buffer; this confirms acceptance, not completion of the asynchronous file write. Exceptions
are caught and reported as FALSE without further logging. The terminal allocation latch is preserved.
Returns FALSE when fatal allocation state is observed before work or after nested calls. The latch remains
set for the caller's task boundary; already accepted or emitted records are not rolled back.
</description>
*)
METHOD TryLogMessage : BOOL
VAR_INPUT
	category : TOF_Core.LOG_CATEGORY;	
END_VAR
VAR_IN_OUT CONSTANT
	message : TOF_Core.ERROR_MESSAGE;
END_VAR
VAR_INPUT
	messageNumber : REFERENCE TO ULINT := 0;
END_VAR
VAR
	textToLog : TOF_Core.ERROR_MESSAGE;
END_VAR
__TRY

	IF TOF_Core.DynamicMemoryManager.HasAllocationFailed THEN
		RETURN;
	END_IF

	IF _MaxRecordsPerFile = TOF_Core.UnsignedInt16.MIN_VALUE
		OR_ELSE _StopRequested
		OR_ELSE _State = SIMPLE_TEXT_FILE_LOGGER_STATE.FAILED
		OR_ELSE _QueueCount >= Parameters.MAX_PENDING_LOG_MESSAGES
	THEN
		TryLogMessage := FALSE;
		RETURN;
	END_IF

	IF __ISVALIDREF(messageNumber) THEN
		textToLog := TOF_Core.WideStrings.Concat255(
			TO_WSTRING(TOF_Core.Exceptions.MESSAGE_NUMBER_PREFIX),
			TO_WSTRING(messageNumber),
			TO_WSTRING(TOF_Core.Exceptions.MESSAGE_NUMBER_SUFFIX)
		);
	END_IF

	TOF_Core.WideStrings.Append255(textToLog, "[", TO_WSTRING(category), "] ");
	TOF_Core.WideStrings.AppendFit(targetString := textToLog, sourceString := message);

	_Queue[_WriteIndex] := textToLog;
	_WriteIndex := _WriteIndex + 1;

	IF _WriteIndex >= Parameters.MAX_PENDING_LOG_MESSAGES THEN
		_WriteIndex := 0;
	END_IF

	_QueueCount := _QueueCount + 1;

	TryLogMessage := TRUE;

	IF TOF_Core.DynamicMemoryManager.HasAllocationFailed THEN
		TryLogMessage := FALSE;
	END_IF

__CATCH
	TryLogMessage := FALSE;
__ENDTRY
END_METHOD

(*!
<summary>Records terminal allocation state without raising or replacing an earlier failure.</summary>
<description>
Returns TRUE when the application fatal latch is observed. Marks the logger FAILED and requests cleanup,
preserving an existing failure diagnostic. No allocation or exception creation occurs. Execute must still
advance already pending I/O before releasing its borrowed buffer; the caller supplies the fatal task boundary.
</description>
*)
METHOD PRIVATE stopAfterAllocationFailure : BOOL
IF NOT TOF_Core.DynamicMemoryManager.HasAllocationFailed THEN
	RETURN;
END_IF

IF _State <> SIMPLE_TEXT_FILE_LOGGER_STATE.FAILED THEN
	_ErrorMessage := "File logger stopped after a terminal allocation failure.";
	_State := SIMPLE_TEXT_FILE_LOGGER_STATE.FAILED;
	_CleanupPending := TRUE;
END_IF

stopAfterAllocationFailure := TRUE;
END_METHOD

END_FUNCTION_BLOCK

// ---- Internal/CurrentNamespace.TcPOU
(*
SPDX-FileCopyrightText: © 2026 Oleksandr Tiutyk <trofimich@gmail.com>
SPDX-License-Identifier: MIT
License: https://opensource.org/license/mit
*)

{attribute 'no_explicit_call' := 'do not call this POU directly'}
PROGRAM INTERNAL CurrentNamespace
VAR
	{attribute 'hide'} 
	_NamespaceExtractor : NamespaceExtractor;
END_VAR

{attribute 'monitoring' := 'call'}
PROPERTY Name : REFERENCE TO STRING
GET
Name REF= _NamespaceExtractor.CurrentNamespace;
END_GET
END_PROPERTY

END_PROGRAM

// ---- Internal/NamespaceExtractor.TcPOU
(*
SPDX-FileCopyrightText: © 2026 Oleksandr Tiutyk <trofimich@gmail.com>
SPDX-License-Identifier: MIT
License: https://opensource.org/license/mit
*)

FUNCTION_BLOCK INTERNAL NamespaceExtractor
VAR_OUTPUT
	{attribute 'init_namespace'} 
	CurrentNamespace : STRING; 	
END_VAR

END_FUNCTION_BLOCK

// ---- QueuedLogger/QueuedLogger.TcPOU
(*
SPDX-FileCopyrightText: © 2026 Oleksandr Tiutyk <trofimich@gmail.com>
SPDX-License-Identifier: MIT
License: https://opensource.org/license/mit
*)

(*!
<summary>Wraps another ILogger and forwards diagnostics from multiple tasks through a bounded queue.</summary>
<description>
Configure once from the cyclic task that will service this instance, before publishing it to logging callers.
Configuration binds Execute to that task; other tasks may enqueue but their Execute calls do nothing. Backend
and wrapper lifetimes must cover all calls and pending processing. Backend is borrowed, not deleted or
configured here; do not call it independently from other tasks or create routing cycles. Queue storage is
fixed by Parameters.QUEUED_LOGGER_CAPACITY. Ordinary text admission does not allocate heap memory; error and
exception formatting may allocate through their existing implementations. A full or unconfigured queue returns
FALSE. TRUE means queued, not written. Errors and exceptions are formatted in the sending task, including
source and local timestamp; aggregate causes become separate records and can interleave with other callers.
Structured backend source fields and backend-specific aggregate markers are not preserved. Plain messages
retain their supplied text. Execute attempts each dequeued record once without retry, even after nonfatal backend FALSE
or exception. FailedDeliveryCount records those failed attempts, not confirmed message loss or durable-write
failures. No callback runs under the queue lock. Queue lock contention may block briefly. All TryLog methods
and Execute contain exceptions and preserve terminal allocation state. PendingMessageCount exposes queued
records only, excluding active delivery and backend work. Stop callers and finish backend processing before
destruction; destruction does not flush pending records. Online-change behavior has not been established.
</description>
*)

{attribute 'no_explicit_call' := 'Use Configure, TryLog methods and Execute'}
FUNCTION_BLOCK FINAL QueuedLogger EXTENDS TOF_Core.Object IMPLEMENTS TOF_Core.ILogger
VAR_STAT
	//! <summary>Static type metadata shared by instances without reading mutable instance state.</summary>
	{attribute 'hide'}
	_ClassName : STRING := __POUNAME();
END_VAR
VAR

	_Backend : TOF_Core.ILogger;
	_OwnerTaskIndex : DINT;
	_QueueLock : Tc2_System.FB_IecCriticalSection;

	_Queue : ARRAY [0..Parameters.QUEUED_LOGGER_CAPACITY - 1] OF QUEUED_LOG_MESSAGE;
	_ReadIndex : UDINT;
	_WriteIndex : UDINT;
	_Count : UDINT;

	_CurrentMessage : QUEUED_LOG_MESSAGE;
	_FailedDeliveryCount : ULINT;
END_VAR

(*!
<summary>Provides the concrete logger type name.</summary>
<description>
Returns borrowed read-only initialized static storage. Reading has no side effects or exceptions.
Do not modify the referenced metadata; initialized storage is available before base initialization.
</description>
*)
{attribute 'monitoring' := 'call'}
PROPERTY ClassName : REFERENCE TO STRING
GET
ClassName REF= _ClassName;
END_GET
END_PROPERTY

(*!
<summary>Assigns the backend and binds processing to the calling cyclic task.</summary>
<description>
Call once before publishing the wrapper. Returns FALSE for null or self backend, non-cyclic context, an
already configured instance or lock failure. No allocation, exception creation or ownership transfer. Does not
initialize the backend or replace an existing configuration.
</description>
<param name="backend">Live logger serviced exclusively through this wrapper; must outlive its use.</param>
*)
METHOD Configure : BOOL
VAR_INPUT
	backend : TOF_Core.ILogger;
END_VAR
VAR
	taskIndex : DINT;
	selfLogger : TOF_Core.ILogger;
END_VAR
taskIndex := TOF_Core.System.GetCurrentTaskIndex();

IF taskIndex < 1 OR_ELSE taskIndex > TOF_Core.System.TASK_COUNT OR_ELSE backend = 0 THEN
	RETURN;
END_IF

selfLogger := THIS^;

IF backend = selfLogger THEN
	RETURN;
END_IF

IF NOT _QueueLock.Enter() THEN
	RETURN;
END_IF

IF _OwnerTaskIndex = 0 THEN
	_Backend := backend;
	_OwnerTaskIndex := taskIndex;
	Configure := TRUE;
END_IF

_QueueLock.Leave();
END_METHOD

(*!
<summary>Services the backend and forwards a bounded batch from the owner task.</summary>
<description>
Other tasks and unconfigured instances do no work. Snapshots the initial queue length and processes at most
that many records, bounded by queue capacity. Calls backend Execute once before forwarding, allowing it to
advance prior work. Each record is removed under the lock and copied into owner-only storage, then forwarded
without the lock. Backend FALSE or exception increments FailedDeliveryCount once without retrying the record
or logging another error. Backend Execute failures and enqueue rejections are excluded. Backend must borrow
the record only for the call and must not reenter this wrapper. Concurrent producers may refill released
slots. Does not guarantee durable output or a fixed execution time; backend and lock latency still apply.
Backend Execute still advances cleanup. Observed fatal allocation state stops further dequeue/delivery,
including after a contained backend failure; the task boundary remains responsible for the fatal raise.
</description>
*)
METHOD Execute
VAR
	taskIndex : DINT;
	messagesToProcess : UDINT;
	i : UDINT;
	lockHeld : BOOL;
	delivered : BOOL;
END_VAR
taskIndex := TOF_Core.System.GetCurrentTaskIndex();

__TRY

	IF NOT _QueueLock.Enter() THEN
		RETURN;
	END_IF

	lockHeld := TRUE;

	IF _OwnerTaskIndex = 0 OR_ELSE taskIndex <> _OwnerTaskIndex THEN
		_QueueLock.Leave();
		lockHeld := FALSE;
		RETURN;
	END_IF

	messagesToProcess := _Count;
	_QueueLock.Leave();
	lockHeld := FALSE;

	__TRY
		_Backend.Execute();
	__CATCH
		// Backend failure must not escape or trigger recursive diagnostics.
	__ENDTRY

	IF TOF_Core.DynamicMemoryManager.HasAllocationFailed THEN
		RETURN;
	END_IF

	FOR i := 1 TO messagesToProcess DO

		IF TOF_Core.DynamicMemoryManager.HasAllocationFailed THEN
			RETURN;
		END_IF

		IF NOT _QueueLock.Enter() THEN
			RETURN;
		END_IF

		lockHeld := TRUE;
		_CurrentMessage := _Queue[_ReadIndex];
		_ReadIndex := _ReadIndex + 1;

		IF _ReadIndex >= Parameters.QUEUED_LOGGER_CAPACITY THEN
			_ReadIndex := 0;
		END_IF

		_Count := _Count - 1;
		_QueueLock.Leave();
		lockHeld := FALSE;

		__TRY

			IF _CurrentMessage.HasMessageNumber THEN
				delivered := _Backend.TryLogMessage(
					category := _CurrentMessage.Category,
					message := _CurrentMessage.Message,
					messageNumber := _CurrentMessage.MessageNumber
				);
			ELSE
				delivered := _Backend.TryLogMessage(category := _CurrentMessage.Category, message := _CurrentMessage.Message);
			END_IF

		__CATCH
			delivered := FALSE;
		__ENDTRY

		IF TOF_Core.DynamicMemoryManager.HasAllocationFailed THEN
			delivered := FALSE;
		END_IF

		IF NOT delivered AND_THEN _FailedDeliveryCount < TOF_Core.UnsignedInt64.MAX_VALUE THEN
			_FailedDeliveryCount := _FailedDeliveryCount + 1;
		END_IF

		IF TOF_Core.DynamicMemoryManager.HasAllocationFailed THEN
			RETURN;
		END_IF

	END_FOR

__CATCH
	IF lockHeld THEN
		_QueueLock.Leave();
	END_IF

__ENDTRY
END_METHOD

(*!
<summary>Counts dequeued records whose delivery failed or observed terminal allocation state.</summary>
<description>
Read from the owner task, or with application-level synchronization against Execute. Updated only by
owner-task Execute. A contained terminal allocation failure counts as a failed attempt even if a hostile
backend returned TRUE. Starts at zero and saturates at UnsignedInt64.MAX_VALUE; no reset is provided. Excludes
enqueue rejection and backend Execute errors. A failed attempt may have produced partial output; successful
acceptance does not guarantee durable storage.
</description>
*)
{attribute 'monitoring' := 'call'}
PROPERTY FailedDeliveryCount : ULINT
GET
FailedDeliveryCount := _FailedDeliveryCount;
END_GET
END_PROPERTY

(*!
<summary>Provides the queued logger NamespaceName.</summary>
<description>Borrowed read-only library namespace.</description>
*)
{attribute 'monitoring' := 'call'}
PROPERTY NamespaceName : REFERENCE TO STRING
GET
NamespaceName REF= CurrentNamespace.Name;
END_GET
END_PROPERTY

(*!
<summary>Returns a synchronized snapshot of the number of records waiting in the queue.</summary>
<description>
Returns -1 if the queue lock cannot be acquired; zero means no queued records at the snapshot instant. Lock
contention may block. Excludes the record currently being forwarded and any work buffered by the backend.
Concurrent producers may change the count immediately after reading. For draining, stop producers and read
from the owner task after Execute returns. Zero does not guarantee successful delivery, completed file I/O or
a closed file. This property does not flush or stop either logger.
</description>
*)
{attribute 'monitoring' := 'call'}
PROPERTY PendingMessageCount : DINT
GET
PendingMessageCount := -1;

IF _QueueLock.Enter() THEN
	PendingMessageCount := TO_DINT(_Count);
	_QueueLock.Leave();
END_IF
END_GET
END_PROPERTY

(*!
<summary>Provides the queued logger SelfSize.</summary>
<description>Size of this concrete instance, including its fixed queue storage.</description>
*)
{attribute 'monitoring' := 'call'}
PROPERTY SelfSize : ULINT
GET
SelfSize := XSIZEOF(THIS^);
END_GET
END_PROPERTY

(*!
<summary>Formats a borrowed error in the sending task and queues its text.</summary>
<description>
Copies source and local timestamp into the text using ERROR.ToString. Retains no reference to ERROR. Returns
FALSE for an invalid reference, failed admission or caught formatting exception. Does not clear terminal
allocation state.
Returns FALSE when fatal allocation state is observed before work or after nested calls. The latch remains
set for the caller's task boundary; already accepted or emitted records are not rolled back.
</description>
<param name="error">Live error formatted during this call.</param>
<param name="messageNumber">Optional number copied with the formatted message.</param>
*)
METHOD TryLogError : BOOL
VAR_INPUT
	error : REFERENCE TO TOF_Core.ERROR;
	messageNumber : REFERENCE TO ULINT := 0;
END_VAR
VAR
	message : TOF_Core.ERROR_MESSAGE;
END_VAR
__TRY

	IF TOF_Core.DynamicMemoryManager.HasAllocationFailed THEN
		RETURN;
	END_IF

	IF NOT __ISVALIDREF(error) THEN
		RETURN;
	END_IF

	message := error.ToString(
		sourceDisplayMode := TOF_Core.ERROR_SOURCE_DISPLAY_MODE.TOP_AND_ROOT,
		timestampDisplayMode := TOF_Core.TIMESTAMP_DISPLAY_MODE.LOCAL
	);
	TryLogError := TryLogMessage(
		category := SEL(
			error.Severity = TOF_Core.ERROR_SEVERITY.CRITICAL,
			TOF_Core.LOG_CATEGORY.ERROR,
			TOF_Core.LOG_CATEGORY.CRITICAL_ERROR
		),
		message := message,
		messageNumber := messageNumber
	);

	IF TOF_Core.DynamicMemoryManager.HasAllocationFailed THEN
		TryLogError := FALSE;
	END_IF

__CATCH
	TryLogError := FALSE;
__ENDTRY
END_METHOD

(*!
<summary>Queues text snapshots of a live exception or its aggregate causes.</summary>
<description>
Formats source and local timestamp before task cleanup. Aggregate causes are visited in stored order and share
the supplied optional request number. Stops on the first failure; already accepted records remain queued and
FALSE may mean partial admission. Concurrent callers may interleave aggregate entries. Empty aggregates are
formatted as ordinary exceptions. Input graphs must be valid and acyclic. No exception reference or clone is
retained; terminal allocation state is preserved.
Returns FALSE when fatal allocation state is observed before work or after nested calls. The latch remains
set for the caller's task boundary; already accepted or emitted records are not rolled back.
</description>
<param name="exception">Live, acyclic exception graph borrowed for formatting.</param>
<param name="severity">Severity used to choose the queued category.</param>
<param name="messageNumber">Optional request number copied to each accepted cause record.</param>
*)
METHOD TryLogException : BOOL
VAR_INPUT
	exception : TOF_Core.IReadOnlyException;
	severity : TOF_Core.ERROR_SEVERITY;
	messageNumber : REFERENCE TO ULINT := 0;
END_VAR
VAR
	message : TOF_Core.ERROR_MESSAGE;
	aggregateException : TOF_Core.IAggregateException;
	innerExceptionCount : UINT;
	i : DINT;
END_VAR
__TRY

	IF TOF_Core.DynamicMemoryManager.HasAllocationFailed THEN
		RETURN;
	END_IF

	IF exception = 0 THEN
		RETURN;
	END_IF

	IF __QUERYINTERFACE(exception, aggregateException) THEN
		innerExceptionCount := aggregateException.InnerExceptionCount;
	END_IF

	IF TOF_Core.DynamicMemoryManager.HasAllocationFailed THEN
		RETURN;
	END_IF

	IF innerExceptionCount > 0 THEN

		FOR i := 0 TO TO_DINT(innerExceptionCount) - 1 DO

			IF TOF_Core.DynamicMemoryManager.HasAllocationFailed THEN
				TryLogException := FALSE;
				RETURN;
			END_IF

			IF NOT THIS^.TryLogException(
				exception := aggregateException.GetInnerException(index := i),
				severity := severity,
				messageNumber := messageNumber
			)
			THEN
				RETURN;
			END_IF

			IF TOF_Core.DynamicMemoryManager.HasAllocationFailed THEN
				TryLogException := FALSE;
				RETURN;
			END_IF

		END_FOR

		TryLogException := TRUE;
	ELSE
		message := exception.GetMessage(showSource := TRUE, timestampDisplayMode := TOF_Core.TIMESTAMP_DISPLAY_MODE.LOCAL);
		TryLogException := TryLogMessage(
			category := SEL(severity = TOF_Core.ERROR_SEVERITY.CRITICAL, TOF_Core.LOG_CATEGORY.ERROR, TOF_Core.LOG_CATEGORY.CRITICAL_ERROR),
			message := message,
			messageNumber := messageNumber
		);
	END_IF

	IF TOF_Core.DynamicMemoryManager.HasAllocationFailed THEN
		TryLogException := FALSE;
	END_IF

__CATCH
	TryLogException := FALSE;
__ENDTRY
END_METHOD

(*!
<summary>Copies one message and its optional number into the bounded queue.</summary>
<description>
Borrows inputs only for this call; the caller must keep them stable while copied. Returns FALSE before
configuration, at capacity, on lock failure or on a caught exception. Commits the entry only after copying its
contents. Does not call the backend or allocate text storage.
Returns FALSE when fatal allocation state is observed before work or after nested calls. The latch remains
set for the caller's task boundary; already accepted or emitted records are not rolled back.
</description>
<param name="category">Category copied into the queued record.</param>
<param name="message">Text copied into owned queue storage.</param>
<param name="messageNumber">Optional borrowed number copied by value.</param>
*)
METHOD TryLogMessage : BOOL
VAR_INPUT
	category : TOF_Core.LOG_CATEGORY;
END_VAR
VAR_IN_OUT CONSTANT
	message : TOF_Core.ERROR_MESSAGE;
END_VAR
VAR_INPUT
	messageNumber : REFERENCE TO ULINT := 0;
END_VAR
VAR
	lockHeld : BOOL;
END_VAR
__TRY

	IF TOF_Core.DynamicMemoryManager.HasAllocationFailed THEN
		RETURN;
	END_IF

	IF NOT _QueueLock.Enter() THEN
		RETURN;
	END_IF

	lockHeld := TRUE;

	IF _OwnerTaskIndex <> 0 AND_THEN _Count < Parameters.QUEUED_LOGGER_CAPACITY THEN
		_Queue[_WriteIndex].Message := message;
		_Queue[_WriteIndex].Category := category;
		_Queue[_WriteIndex].HasMessageNumber := __ISVALIDREF(messageNumber);

		IF _Queue[_WriteIndex].HasMessageNumber THEN
			_Queue[_WriteIndex].MessageNumber := messageNumber;
		END_IF

		_WriteIndex := _WriteIndex + 1;

		IF _WriteIndex >= Parameters.QUEUED_LOGGER_CAPACITY THEN
			_WriteIndex := 0;
		END_IF

		_Count := _Count + 1;
		TryLogMessage := TRUE;
	END_IF

	_QueueLock.Leave();
	lockHeld := FALSE;

	IF TOF_Core.DynamicMemoryManager.HasAllocationFailed THEN
		TryLogMessage := FALSE;
	END_IF

__CATCH
	IF lockHeld THEN
		_QueueLock.Leave();
	END_IF

	TryLogMessage := FALSE;
__ENDTRY
END_METHOD

END_FUNCTION_BLOCK

// ---- EventLogger/EventLogger.TcPOU
(*
SPDX-FileCopyrightText: © 2026 Oleksandr Tiutyk <trofimich@gmail.com>
SPDX-License-Identifier: MIT
License: https://opensource.org/license/mit
*)

(*!
<summary>Writes diagnostics through TwinCAT EventLogger and expands aggregate exceptions into entries.</summary>
<description>
Provide one live event definition per category with a message placeholder {0}; the native event definition
determines event identity and severity. Constructor arguments are copied, not borrowed. No later
configuration API or native online-change handoff is provided. Keep initialization/destruction separate
from application calls; derived implementations must preserve these lifetime and no-throw guarantees.
Use this backend for TwinCAT EventLogger events with structured source information when logging errors and
exceptions directly. Use one task for direct calls on each instance without same-instance reentry; concurrent use of its internal
FB_TcEventLogger has no established guarantee here. For callers in multiple tasks, use QueuedLogger and let
only its owner task access this backend; do not bypass the wrapper with concurrent direct calls. QueuedLogger
forwards text records, so exception source is included in text rather than the structured source field, and
backend-specific aggregate formatting is not preserved. Execute performs no cyclic work. Exception logging
accepts IReadOnlyException and reads borrowed diagnostics without transferring ownership. Implementations must
not retain exception references beyond their task cleanup. Numbered messages preserve the number and truncate
oversized text to ERROR_MESSAGE capacity with a final ellipsis. TryLog methods must satisfy the no-throw
contract even when called directly, without LogManager. Does not propagate exceptions, including failures
while reading or formatting diagnostics and calling the backend; returns FALSE instead. Already emitted
entries are not rolled back, so FALSE may follow partial output. Caught exceptions are not logged again. The
fatal allocation latch is preserved for RaiseIfAllocationFailed at the task boundary outside recoverable
handlers.
</description>
*)

{attribute 'no_explicit_call' := 'do not call this function block directly'}
FUNCTION_BLOCK EventLogger EXTENDS TOF_Core.Object IMPLEMENTS TOF_Core.ILogger
VAR_STAT
	//! <summary>Static type metadata shared by instances without reading mutable instance state.</summary>
	{attribute 'hide'} 
	_ClassName : STRING := __POUNAME();
END_VAR
VAR
	
	_EventLogger : Tc3_EventLogger.FB_TcEventLogger;
	
	_DebugEventType : Global.TcEventEntry;
	_InformationEventType : Global.TcEventEntry;
	_WarningEventType : Global.TcEventEntry;
	_ErrorEventType : Global.TcEventEntry;
	_CriticalErrorEventType : Global.TcEventEntry;	
END_VAR

(*!
<summary>Provides the concrete logger type name.</summary>
<description>
Returns borrowed read-only initialized static storage. Reading has no side effects or exceptions.
Do not modify the referenced metadata; initialized storage is available before base initialization.
</description>
*)
{attribute 'monitoring' := 'call'}
PROPERTY ClassName : REFERENCE TO STRING
GET
ClassName REF= _ClassName;
END_GET
END_PROPERTY

(*!
<summary>Completes without work because this logger has no cyclic processing.</summary>
<description>Does not raise exceptions.</description>
*)
METHOD Execute
// EventLogger has no cyclic work
END_METHOD

(*!
<summary>FB_Init is always available implicitly and it is used primarily for initialization.</summary>
<description>
The return value is not evaluated. Assigns and retains event definitions for each severity category.
</description>
<param name="debugEventType">Event entry used for DEBUG category.</param>
<param name="informationEventType">Event entry used for INFORMATION category.</param>
<param name="warningEventType">Event entry used for WARNING category.</param>
<param name="errorEventType">Event entry used for ERROR category.</param>
<param name="criticalErrorEventType">Event entry used for CRITICAL_ERROR category.</param>
*)
METHOD FB_Init: BOOL
VAR_INPUT
	bInitRetains : BOOL; // TRUE: the retain variables are initialized (reset warm / reset cold)
	bInCopyCode : BOOL;  // TRUE: the instance will be copied to the copy code afterward (online change)
	debugEventType : Global.TcEventEntry;
	informationEventType : Global.TcEventEntry;
	warningEventType : Global.TcEventEntry;
	errorEventType : Global.TcEventEntry;
	criticalErrorEventType : Global.TcEventEntry;
END_VAR
_DebugEventType := debugEventType;	
_InformationEventType := informationEventType;
_WarningEventType := warningEventType;
_ErrorEventType := errorEventType;
_CriticalErrorEventType := criticalErrorEventType;
END_METHOD

(*!
<summary>Sends a diagnostic with its source and optional message number.</summary>
<description>
When a number is supplied, preserves the number prefix and as much message text as fits ERROR_MESSAGE.
Truncated text ends with U+2026. Formatting uses local storage and does not raise a size-overflow exception.
Returns FALSE for an unsupported category or failed send.
Contains formatting and native exceptions in this frame so local native FB instances exit normally.
Returns FALSE when fatal allocation state is observed before work or after nested calls. The latch remains
set for the caller's task boundary; already accepted or emitted records are not rolled back.
</description>
*)
METHOD PROTECTED InternalTryLogMessage : BOOL
VAR_INPUT
	category : TOF_Core.LOG_CATEGORY;	
END_VAR
VAR_IN_OUT CONSTANT
	message : TOF_Core.ERROR_MESSAGE;
END_VAR
VAR_INPUT
	source : Tc2_System.T_MaxString;
	messageNumber : REFERENCE TO ULINT := 0;
END_VAR
VAR	
	sourceInfo : Tc3_EventLogger.FB_TcSourceInfo;
	arguments : Tc3_EventLogger.FB_TcArguments;
	messageWithNumber : TOF_Core.ERROR_MESSAGE;
	methodResult : HRESULT;
END_VAR
__TRY

	IF TOF_Core.DynamicMemoryManager.HasAllocationFailed THEN
		RETURN;
	END_IF

	sourceInfo.sName := source;

	IF __ISVALIDREF(messageNumber) THEN
		messageWithNumber := TOF_Core.WideStrings.Concat255(
			TO_WSTRING(TOF_Core.Exceptions.MESSAGE_NUMBER_PREFIX),
			TO_WSTRING(messageNumber),
			TO_WSTRING(TOF_Core.Exceptions.MESSAGE_NUMBER_SUFFIX)
		);
		TOF_Core.WideStrings.AppendFit(targetString := messageWithNumber, sourceString := message);
		arguments.AddWString(value := messageWithNumber);
	ELSE
		arguments.AddWString(value := message);
	END_IF

	IF TOF_Core.DynamicMemoryManager.HasAllocationFailed THEN
		RETURN;
	END_IF

	CASE category OF
		TOF_Core.LOG_CATEGORY.DEBUG:
			methodResult := _EventLogger.SendMessageEx(
				stEventEntry := _DebugEventType,
				ipSourceInfo := sourceInfo,
				nTimeStamp := 0,
				ipArguments := arguments
			);

		TOF_Core.LOG_CATEGORY.INFORMATION:
			methodResult := _EventLogger.SendMessageEx(
				stEventEntry := _InformationEventType,
				ipSourceInfo := sourceInfo,
				nTimeStamp := 0,
				ipArguments := arguments
			);

		TOF_Core.LOG_CATEGORY.WARNING:
			methodResult := _EventLogger.SendMessageEx(
				stEventEntry := _WarningEventType,
				ipSourceInfo := sourceInfo,
				nTimeStamp := 0,
				ipArguments := arguments
			);

		TOF_Core.LOG_CATEGORY.ERROR:
			methodResult := _EventLogger.SendMessageEx(
				stEventEntry := _ErrorEventType,
				ipSourceInfo := sourceInfo,
				nTimeStamp := 0,
				ipArguments := arguments
			);

		TOF_Core.LOG_CATEGORY.CRITICAL_ERROR:
			methodResult := _EventLogger.SendMessageEx(
				stEventEntry := _CriticalErrorEventType,
				ipSourceInfo := sourceInfo,
				nTimeStamp := 0,
				ipArguments := arguments
			);

		ELSE
			Tc2_System.ADSLOGSTR(
				msgCtrlMask := Tc2_System.Global_Variables.ADSLOG_MSGTYPE_ERROR OR Tc2_System.Global_Variables.ADSLOG_MSGTYPE_LOG,
				msgFmtStr := Tc2_Standard.CONCAT(STR1 := 'Unsupported log category ', STR2 := TO_STRING(category)),
				strArg := ''
			);

			RETURN;
	END_CASE

	IF TOF_Core.DynamicMemoryManager.HasAllocationFailed THEN
		RETURN;
	END_IF

	IF Tc3_Module.FAILED(hr := methodResult) THEN
		Tc2_System.ADSLOGSTR(
			msgCtrlMask := Tc2_System.Global_Variables.ADSLOG_MSGTYPE_ERROR OR Tc2_System.Global_Variables.ADSLOG_MSGTYPE_LOG,
			msgFmtStr := Tc2_Standard.CONCAT(
				STR1 := 'FB_TcMessage creation failed with HRESULT = ',
				STR2 := TO_STRING(methodResult)
			),
			strArg := ''
		);

		RETURN;
	END_IF

	InternalTryLogMessage := TRUE;

	IF TOF_Core.DynamicMemoryManager.HasAllocationFailed THEN
		InternalTryLogMessage := FALSE;
	END_IF

__CATCH
	// Contain failure before local native argument/source objects leave this frame.
	InternalTryLogMessage := FALSE;
__ENDTRY
END_METHOD

(*!
<summary>Borrows the library namespace.</summary>
<description>
Read-only compiler-initialized storage; do not modify the referenced text.
</description>
*)
{attribute 'monitoring' := 'call'}
PROPERTY NamespaceName : REFERENCE TO STRING
GET
NamespaceName REF= CurrentNamespace.Name;
END_GET
END_PROPERTY

(*!
<summary>Reports the size of this concrete event logger instance.</summary>
<description>
The result includes embedded native state but excludes allocations owned internally by native services.
</description>
*)
{attribute 'monitoring' := 'call'}
PROPERTY SelfSize : ULINT
GET
SelfSize := XSIZEOF(THIS^);
END_GET
END_PROPERTY

(*!
<summary>Attempts to log a borrowed error without propagating exceptions.</summary>
<description>
Borrows inputs only for the call. TRUE reports backend acceptance, not guaranteed durable storage. Does not
propagate exceptions, including failures while reading or formatting diagnostics and calling the backend;
returns FALSE instead. Already emitted entries are not rolled back, so FALSE may follow partial output. Caught
exceptions are not logged again. The fatal allocation latch is preserved for RaiseIfAllocationFailed at the
task boundary outside recoverable handlers.
Returns FALSE when fatal allocation state is observed before work or after nested calls. The latch remains
set for the caller's task boundary; already accepted or emitted records are not rolled back.
</description>
*)
METHOD TryLogError : BOOL
VAR_INPUT
	error : REFERENCE TO TOF_Core.ERROR;
	messageNumber : REFERENCE TO ULINT := 0;
END_VAR
VAR
	message : TOF_Core.ERROR_MESSAGE;
END_VAR
__TRY

	IF TOF_Core.DynamicMemoryManager.HasAllocationFailed THEN
		RETURN;
	END_IF

	IF NOT __ISVALIDREF(error) THEN
		RETURN;
	END_IF

	message := error.ToString(
		sourceDisplayMode := TOF_Core.ERROR_SOURCE_DISPLAY_MODE.HIDDEN,
		timestampDisplayMode := TOF_Core.TIMESTAMP_DISPLAY_MODE.HIDDEN
	);

	IF TOF_Core.DynamicMemoryManager.HasAllocationFailed THEN
		RETURN;
	END_IF

	TryLogError := InternalTryLogMessage(
		category := SEL(
			error.Severity = TOF_Core.ERROR_SEVERITY.CRITICAL,
			TOF_Core.LOG_CATEGORY.ERROR,
			TOF_Core.LOG_CATEGORY.CRITICAL_ERROR
		),
		message := message,
		source := error.GetSource(appendRootSource := TRUE),
		messageNumber := messageNumber
	);

	IF TOF_Core.DynamicMemoryManager.HasAllocationFailed THEN
		TryLogError := FALSE;
	END_IF

__CATCH
	TryLogError := FALSE;
__ENDTRY
END_METHOD

(*!
<summary>Attempts to log diagnostic information from a read-only exception view.</summary>
<description>
Borrows the exception for the call without clearing it or taking ownership. The exception and its inner causes
must remain live and form an acyclic graph while their diagnostics are read. Nonempty aggregates produce
separate entries in stored order, sharing the optional request number. Nonfatal FALSE does not suppress later
entries; a thrown diagnostic failure or observed terminal allocation state stops further processing. Logging does not extend their lifetime. Does not propagate
exceptions, including failures while reading or formatting diagnostics and calling the backend; returns FALSE
instead. Already emitted entries are not rolled back, so FALSE may follow partial output. Caught exceptions
are not logged again. The fatal allocation latch is preserved for RaiseIfAllocationFailed at the task boundary
outside recoverable handlers.
Returns FALSE when fatal allocation state is observed before work or after nested calls. The latch remains
set for the caller's task boundary; already accepted or emitted records are not rolled back.
</description>
<param name="exception">Exception view to read; null is ignored.</param>
<param name="severity">Severity used to select the log category.</param>
*)
METHOD TryLogException : BOOL
VAR_INPUT
	exception : TOF_Core.IReadOnlyException;
	severity : TOF_Core.ERROR_SEVERITY;
	messageNumber : REFERENCE TO ULINT := 0;
END_VAR
VAR
	message : TOF_Core.ERROR_MESSAGE;
	aggregateException : TOF_Core.IAggregateException;
	innerExceptionCount : UINT;
	i : DINT;
END_VAR
__TRY

	IF TOF_Core.DynamicMemoryManager.HasAllocationFailed THEN
		RETURN;
	END_IF

	IF exception = 0 THEN
		RETURN;
	END_IF

	IF __QUERYINTERFACE(exception, aggregateException) THEN
		innerExceptionCount := aggregateException.InnerExceptionCount;
	END_IF

	IF TOF_Core.DynamicMemoryManager.HasAllocationFailed THEN
		RETURN;
	END_IF

	IF innerExceptionCount = 0 THEN
		message := exception.GetMessage(showSource := FALSE, timestampDisplayMode := TOF_Core.TIMESTAMP_DISPLAY_MODE.LOCAL);

		IF TOF_Core.DynamicMemoryManager.HasAllocationFailed THEN
			RETURN;
		END_IF

		TryLogException := InternalTryLogMessage(
			category := SEL(severity = TOF_Core.ERROR_SEVERITY.CRITICAL, TOF_Core.LOG_CATEGORY.ERROR, TOF_Core.LOG_CATEGORY.CRITICAL_ERROR),
			message := message,
			source := exception.GetSourceDescription(),
			messageNumber := messageNumber
		);
	ELSE
		TryLogException := TRUE;

		FOR i := 0 TO TO_DINT(innerExceptionCount) - 1 DO

			IF TOF_Core.DynamicMemoryManager.HasAllocationFailed THEN
				TryLogException := FALSE;
				RETURN;
			END_IF

			TryLogException := TryLogException AND THIS^.TryLogException(
				exception := aggregateException.GetInnerException(index := i),
				severity := severity,
				messageNumber := messageNumber
			);

			IF TOF_Core.DynamicMemoryManager.HasAllocationFailed THEN
				TryLogException := FALSE;
				RETURN;
			END_IF

		END_FOR

	END_IF

	IF TOF_Core.DynamicMemoryManager.HasAllocationFailed THEN
		TryLogException := FALSE;
	END_IF

__CATCH
	TryLogException := FALSE;
__ENDTRY
END_METHOD

(*!
<summary>Attempts to log borrowed message text without propagating exceptions.</summary>
<description>
Borrows inputs only for the call. TRUE reports backend acceptance, not guaranteed durable storage. Does not
propagate exceptions, including failures while reading or formatting diagnostics and calling the backend;
returns FALSE instead. Already emitted entries are not rolled back, so FALSE may follow partial output. Caught
exceptions are not logged again. The fatal allocation latch is preserved for RaiseIfAllocationFailed at the
task boundary outside recoverable handlers.
Returns FALSE when fatal allocation state is observed before work or after nested calls. The latch remains
set for the caller's task boundary; already accepted or emitted records are not rolled back.
</description>
*)
METHOD TryLogMessage : BOOL
VAR_INPUT
	category : TOF_Core.LOG_CATEGORY;	
END_VAR
VAR_IN_OUT CONSTANT
	message : TOF_Core.ERROR_MESSAGE;
END_VAR
VAR_INPUT
	messageNumber : REFERENCE TO ULINT := 0;
END_VAR
__TRY

	IF TOF_Core.DynamicMemoryManager.HasAllocationFailed THEN
		RETURN;
	END_IF

	TryLogMessage := InternalTryLogMessage(category := category, message := message, source := '', messageNumber := messageNumber);

	IF TOF_Core.DynamicMemoryManager.HasAllocationFailed THEN
		TryLogMessage := FALSE;
	END_IF

__CATCH
	TryLogMessage := FALSE;
__ENDTRY
END_METHOD

END_FUNCTION_BLOCK
